//==================================================================================================
//							Beckhoff Automation Poland
//									3.01.2022
//	Function block running home procedure in torque mode
//	Avaliable two modes:
//	1. Lag based - bLagBased = TRUE - define lrLagLimit which decides about end of movement
//	2. Torque based - bLagBased = FALSE - define lrTorqueLimit and lrTorqueTolerance which decides about end of movement
//
//	Library: Tc3_MC2_AdvancedHoming, Tc2_MC2, 
//
//  v1.0	|| TC v 3.1.4024.22		|| First edition 
//==================================================================================================
FUNCTION_BLOCK FB_HomingTorque_1
VAR_IN_OUT
	Axis 										: Tc2_MC2.AXIS_REF;
END_VAR  
VAR_INPUT
	bExecute									: BOOL;					// The command is executed with a rising edge.
	bLagBased									: BOOL;					// TRUE: MC_StepBlockLagBased, FALSE: MC_StepBlock
	eDirection									: Tc3_MC2_AdvancedHoming.MC_Home_Direction;	// 
	lrVelocity									: LREAL;				// Maximum travel velocity (>0)
	lrSetPosition								: LREAL;				// Position value to which the axis position is to be set. 
	lrDetectionVelocityLimit					: LREAL;				// Velocity that must be fallen below for the time DetectionVelocityTime in order to detect driving against the fixed stop.
	tDetectionVelocityTime						: TIME;					// Time for detecting the velocity undershoot when driving against the fixed stop.
	tTimeLimit									: TIME;					// Exceeding this time leads to the search procedure being aborted.
	lrDistanceLimit								: LREAL;				// Exceeding this distance in relation to the start position leads to the search procedure being aborted.
	lrTorqueLimit								: LREAL;				// The motor torque is limited to this value, in relation to the weight counterbalance that is possibly parameterized in the drive, in order to avoid mechanical damage.
	lrTorqueTolerance							: LREAL;				// Tolerance related to the TorqueLimit within which driving against the fixed stop is detected.
	lrLagLimit									: LREAL;				// Position lag value which, if exceeded, leads to detection of driving against the fixed stop.
	lrDistance									: LREAL;				// Distance by which the axis moves away from the current position.
END_VAR                             		
VAR_OUTPUT                              		
	bDone										: BOOL;
	bBusy										: BOOL;
	bCommandAborted								: BOOL;
	bError										: BOOL;
	nErrorID									: UDINT;
END_VAR
VAR
//=========================== Common ============================
	nStep										: UDINT;
	stParameter									: Tc3_MC2_AdvancedHoming.MC_HomingParameter;
	stOptions									: Tc3_MC2_AdvancedHoming.ST_Home_Options3;
//========================= Step Block ==========================
	mcStepBlock									: Tc3_MC2_AdvancedHoming.MC_StepBlock;
	mcStepBlockLag								: Tc3_MC2_AdvancedHoming.MC_StepBlockLagBased;
//=========================== Finish ============================
	mcFinishHoming								: Tc3_MC2_AdvancedHoming.MC_FinishHoming;
//============================ Abort ============================
	mcAbortHoming								: Tc3_MC2_AdvancedHoming.MC_AbortHoming;
//========================== Internal ===========================
    {attribute 'hide'}
	nErrorID_Int								: UDINT;
//===============================================================
END_VAR

//====== Call FBs outside CASE - easier debugging ===============
mcStepBlockLag(Axis								:= Axis, 
				Parameter						:= stParameter);
				                        		
mcStepBlock(	Axis							:= Axis, 
				Parameter						:= stParameter);	
                                        		
mcFinishHoming(	Axis							:= Axis, 
				Parameter						:= stParameter);
				                        	
mcAbortHoming(	Axis							:= Axis, 
				Parameter						:= stParameter);
				
//============== CASE instruction - step machine ================
CASE nStep OF
	
	0: // Wait for command
	
		IF bExecute THEN
			bBusy								:= TRUE;
			// Latch finish parameters
			mcFinishHoming.Distance				:= lrDistance;
			mcFinishHoming.Velocity				:= lrVelocity;
				
			IF bLagBased THEN

				mcStepBlockLag(Axis				:= Axis, 
						Parameter				:= stParameter, 
						Execute					:= TRUE, 
						Direction				:= eDirection, 
						Velocity				:= lrVelocity,
						SetPosition				:= lrSetPosition, 
						DetectionVelocityLimit	:= lrDetectionVelocityLimit, 
						DetectionVelocityTime	:= tDetectionVelocityTime, 
						TimeLimit				:= tTimeLimit, 
						DistanceLimit			:= lrDistanceLimit, 
						TorqueLimit				:= lrTorqueLimit, 
						LagLimit				:= lrLagLimit, 
						Options					:= stOptions);
				
				nStep							:= 1000;
				
			ELSE

				mcStepBlock(Axis				:= Axis, 
						Parameter				:= stParameter, 
						Execute					:= TRUE, 
						Direction				:= eDirection, 
						Velocity				:= lrVelocity,
						SetPosition				:= lrSetPosition, 
						DetectionVelocityLimit	:= lrDetectionVelocityLimit, 
						DetectionVelocityTime	:= tDetectionVelocityTime, 
						TimeLimit				:= tTimeLimit, 
						DistanceLimit			:= lrDistanceLimit, 
						TorqueLimit				:= lrTorqueLimit, 
						TorqueTolerance			:= lrTorqueTolerance, 
						Options					:= stOptions);
						
				nStep							:= 2000;
				
			END_IF
		END_IF
	
	1000: // Wait till end
	
		IF mcStepBlockLag.Done THEN
			mcStepBlockLag.Execute				:= FALSE;
			nStep 								:= 3000;
		END_IF
		
		IF mcStepBlockLag.CommandAborted THEN
			mcStepBlockLag.Execute				:= FALSE;
			bBusy 								:= FALSE;
			bCommandAborted						:= TRUE;
			nStep 								:= 6000;
		END_IF
		
		IF mcStepBlockLag.Error THEN
			mcStepBlockLag.Execute				:= FALSE;
			nErrorID_Int						:= mcStepBlockLag.ErrorID;
			nStep 								:= 4000;
		END_IF
	
	2000: // Wait till end
	
		IF mcStepBlock.Done THEN
			mcStepBlock.Execute					:= FALSE;
			nStep 								:= 3000;
		END_IF
		
		IF mcStepBlock.CommandAborted THEN
			mcStepBlock.Execute					:= FALSE;
			bBusy 								:= FALSE;
			bCommandAborted						:= TRUE;
			nStep 								:= 6000;
		END_IF
		
		IF mcStepBlock.Error THEN
			mcStepBlock.Execute					:= FALSE;
			nErrorID_Int						:= mcStepBlock.ErrorID;
			nStep 								:= 4000;
		END_IF
		
	3000: // MC_FinishHoming
	
		mcFinishHoming.Execute					:= TRUE;				
		nStep									:= nStep + 10;
		
	3010: // Wait till end
	
		IF mcFinishHoming.Done THEN
			mcFinishHoming.Execute				:= FALSE;
			bBusy 								:= FALSE;
			bDone 								:= TRUE;
			nStep 								:= 5000;
		END_IF
		
		IF mcFinishHoming.CommandAborted THEN
			mcFinishHoming.Execute				:= FALSE;
			bBusy 								:= FALSE;
			bCommandAborted						:= TRUE;
			nStep 								:= 6000;
		END_IF
		
		IF mcFinishHoming.Error THEN
			mcFinishHoming.Execute				:= FALSE;
			bBusy 								:= FALSE;
			bError								:= TRUE;
			nErrorID							:= mcFinishHoming.ErrorID;
			nStep 								:= 10000;
		END_IF	
		
	4000: // MC_AbortHoming
	
		mcAbortHoming.Execute					:= TRUE;				
		nStep									:= nStep + 10;
		
	4010: // Wait till end
	
		// No matter what is the end, we go to error State
		IF NOT mcAbortHoming.Busy THEN
			mcAbortHoming.Execute				:= FALSE;
			bBusy 								:= FALSE;
			bError								:= TRUE;
			nErrorID							:= nErrorID_Int;			
			nStep								:= 10000;
		END_IF
		
	5000: // Done
		
		bDone									:= bExecute;
		IF NOT bExecute THEN
			nStep 								:= 0;
		END_IF	
	
	6000: // Command Aborted
	
		bCommandAborted							:= bExecute;
		IF NOT bExecute THEN
			nStep 								:= 0;
		END_IF
		
	10000..20000: // Error
	
		bError									:= bExecute;
		IF NOT bExecute THEN
			nErrorID							:= 0;
			nErrorID_Int						:= 0;
			nStep 								:= 0;
		END_IF
		
END_CASE
//===============================================================

END_FUNCTION_BLOCK

(* stored: Version 1.2.0.0, ProductVersion 3.1.4026.13, FileIdentifier 7a2245a8337ed4cc9486d3fbe3d0acdadc9609b8, FileSignature 812740f9a43f656abcc81213823e7939bd4097e279d62f975c116d526fbecc32e6ad33b12523b0f14f692e6324c7a8f665506190bc8a6ceb26ab2617bf901301df4fad02c06319a660af28e2c7e81577af5a839ed34885ad980301db6d4ee6a02821be07e070bc4919e916830c8da9153e4f23a18f2a52200badd1225c91717b098191bd93ad0bd8130b764211ac88b010037cdc6d273186b72108d6252580d914410cf7a41b0cbd2e09b1d85a42d5ef448c62aac05144f201d3fcffd099e0b419d5d901d71e3f987f65a4963996f276e0827c5b536c127d4c9fa34f6325e4982fa416d5317adf527c8d940e2ede4f86cb6114d74e64d9be0332e25a01425dfb
   POU FB_HomingTorque_1: Id {354dae90-8779-4645-b25f-1a2f762786fa}, SpecialFunc None *)
